{attribute 'qualified_only'}
VAR_GLOBAL
	Points		: ARRAY[0..9] OF ST_Point;
END_VAR

(* stored: Version 1.1.0.1, ProductVersion 3.1.4024.12
   GVL GVL: Id {4dae7c4f-42d7-45a0-8f83-864bd15eb14f} *)
